TYPE ST_PQVoltageData EXTENDS ST_PQPowerData:
STRUCT
	b_VoltagesOK			: 	BOOL;
	e_ACrotationStatus		:	eACRotationState;
	ar_PhaseVoltage			: 	ARRAY[0..3] OF REAL;
	ar_LineVoltage			:	ARRAY[0..3] OF REAL;
	ar_Frequency			: 	ARRAY[0..3] OF REAL;
	r_VoltageUnbalance		: 	REAL;
	ar_VoltageTHD			: 	ARRAY[0..3] OF REAL;
END_STRUCT
END_TYPE

(* stored: Version 1.1.0.1, ProductVersion 3.1.4026.18
   DUT ST_PQVoltageData: Id {ea032aac-7c32-46dd-9283-7e1b9d3b84d4} *)
